Fanuc KAREL source: kd00041.KL

-- PROVISIONAL review KL for V770-1; original PC SHA256 959f92d068033a269f001d5ee0ddbe71a82655bd5228d540ed7e877186196932
-- Incomplete behavior may be omitted. Consult companion uncertainty JSON. Do not deploy.
PROGRAM KD00041
%NOLOCKGROUP
BEGIN
  -- UNRESOLVED_PC offsets 5-12; opcodes 9D,23
  -- UNRESOLVED_PC offsets 17-21; opcodes 7F
END KD00041
